{attribute 'GeneratedUsingTerminal: EL3681-0000-0018'}
{attribute addProperty BoxType "EL3681-0000-0018"}
{attribute addProperty Id "SAI_InputsAT %I*SAI_Inputs_84B29FE914SAI_RangeAT %I*SAI_Range_BDBF6DA92SAI_Range_1AT %Q*SAI_Range_2A187FC54WcStateAT %I*WcState_9091E0EB2InfoDataAT %I*InfoData_94A18F5E2"}
{attribute addProperty CRC "3724011598"}
{attribute addProperty Size "24"}
TYPE EL3681_DDF7E84E EXTENDS EtcSlaveTerminalBase_947E5A46 :
STRUCT
	{attribute addProperty Name "SAI_Inputs"}
	SAI_Inputs : SAI_Inputs_84B29FE9;
	{attribute addProperty Name "SAI_Range"}
	SAI_Range : SAI_Range_BDBF6DA9;
	{attribute addProperty Name "SAI_Range_1"}
	SAI_Range_1 : SAI_Range_2A187FC5;
	{attribute addProperty Name "WcState"}
	WcState : WcState_9091E0EB;
	{attribute addProperty Name "InfoData"}
	InfoData : InfoData_94A18F5E;
END_STRUCT
END_TYPE

(* stored: Version 1.2.0.0, ProductVersion 3.1.4024.9
   DUT EL3681_DDF7E84E: Id {7c4ea5f0-c5af-43f4-af4b-7b0a45bf6c33} *)
